{attribute addProperty BoxType "EL3602-0020-0018"}
{attribute addProperty Id "AI_Inputs_ChannelAT %I*ARRAY[0..1] OF AI_Inputs_Channel_0A6FB19B19424.250WcStateAT %I*WcState_98A4DF7520.250InfoDataAT %I*InfoData_BC63D37F80100"}
{attribute addProperty CRC "3593633689"}
{attribute addProperty SizeInBites "276"}
{attribute addProperty SizeInBytes "34.5"}
TYPE EL3602_5DBFB1A0 :
STRUCT
	{attribute addProperty Name "AI_Inputs_Channel"}
	AI_Inputs_Channel : ARRAY[0..1] OF AI_Inputs_Channel_0A6FB19B;
	{attribute addProperty Name "WcState"}
	WcState : WcState_98A4DF75;
	{attribute addProperty Name "InfoData"}
	InfoData : InfoData_BC63D37F;
END_STRUCT
END_TYPE

(* stored: Version 1.2.0.0, ProductVersion 3.1.4024.9
   DUT EL3602_5DBFB1A0: Id {aa6cf93f-b704-4792-bb11-86fb37458c57} *)
